// TIA Portal V17 export
// export: Created 2023-02-14T02:49:48.6840805Z, ExportSetting WithDefaults, DisplayName Totally Integrated Automation Portal, DisplayVersion V17, DisplayName TIA Portal Openness, DisplayVersion V17, DisplayName TIA Portal Teamcenter Gateway, DisplayVersion V17, DisplayName TIA Portal Version Control Interface, DisplayVersion V17, DisplayName SINAMICS Startdrive Advanced, DisplayVersion V17, DisplayName SINAMICS Startdrive G130, G150, S120, S150, SINAMICS MV, S210, DisplayVersion V17, DisplayName SINAMICS Startdrive G110M, G120, G120C, G120D, G120P, G115D, DisplayVersion V17, DisplayName STEP 7 Professional, DisplayVersion V17, DisplayName STEP 7 Safety, DisplayVersion V17, DisplayName WinCC Professional, DisplayVersion V17
FUNCTION_BLOCK "BFT_Type2"   // FB352, LAD
{ S7_Optimized_Access := 'TRUE' }
VERSION : 0.1
// Buffer Tank with Agitator
// stored: AutoNumber false, IsIECCheckEnabled false, IsRetainMemResEnabled false, MemoryReserve 100, SetENOAutomatically false, UDAEnableTagReadback false
   VAR_INPUT
      "IN_FBAV.01" : Bool := FALSE;   // Tank Flushing Water Valve
      "IN_FBAV.02" : Bool := FALSE;   // Tank CIP Top Inlet Valve
      "IN_FBAV.03" : Bool := FALSE;   // Tank Tank Outlet Valve
      "IN_FBAV.04" : Bool := FALSE;   // Tank CIP Return Valve
      "IN_FBAV.05" : Bool := FALSE;   // Tank Inlet Vinegar Valve
      "IN_FBAV.06" : Bool := FALSE;   // Tank CIP Valve
      "IN_FBAV.07" : Bool := FALSE;   // Tank CIP Valve
      "IN_FBAV.08" : Bool := FALSE;   // Line CIP Bypass Valve
      "IN_FBAV.09" : Bool := FALSE;   // Line CIP Valve
      "IN_FBAV.10" : Bool;   // Tank Inlet Valve
      "IN_FBAV.11" : Bool;   // Line CIP Valve
      "IN_FBAV.12" : Bool;   // Line CIP Valve
      IN_LT01 : Real;   // Tank Level Transmitter
      "IN_FBP.01" : Bool := FALSE;   // Transfer Pump
      "IN_P.01-Speed" : Real;   // Transfer Pump AV Speed
      "IN_FBP.02" : Bool := FALSE;   // CIP Pump
      "IN_P.02-Speed" : Real;   // CIP Pump AV Speed
      "IN_FBP.03" : Bool := FALSE;   // Supply Pump
      "IN_P.03-Speed" : Real;   // Supply Pump AV Speed
      IN_FBXA : Bool := FALSE;   // Agitator
      "IN_XA-Speed" : Real;   // Agitator AV Speed
      DosePumpSpeed : Real;
      "DoseON-OFF" : Bool := FALSE;
      "DosePumpON-OFF" : Bool := FALSE;
      CIPPulse : Bool := FALSE;
      CIP_Supply_ON : Bool;
      CIP_Busy : Bool;   // Line CIP in USE
      LineTrf_OK : Bool := FALSE;
      LineFlush_OK : Bool;
      Loading_Busy : Bool;   // Other tank at loading
      LCS_Start : Bool;   // Start Command from LCS
      LCS_Stop : Bool;   // Stop Command from LCS
      LCS_Dose : Bool;   // Start dose command from LCS
      InloadDose_AV : Bool;   // Inload Dose Valve Open
      InloadDose_P : Bool;   // Inload Dose Pump Running
      CountMode : Bool;   // 0 = Pulse Counting, 1 = Real Count
      FT_Pulse : Bool;   // Pulse Flow Meter
      FT_Total : Real;   // Inload Dose Actual Value
      IN_LDT : Date_And_Time;
   END_VAR
   VAR_OUTPUT
      "OUT_AV.01" : Bool := FALSE;   // Tank Flushing Water Valve
      "OUT_AV.02" : Bool := FALSE;   // Tank CIP Top Inlet Valve
      "OUT_AV.03" : Bool := FALSE;   // Tank Tank Outlet Valve
      "OUT_AV.04" : Bool := FALSE;   // Tank CIP Return Valve
      "OUT_AV.05" : Bool := FALSE;   // Tank Inlet Vinegar Valve
      "OUT_AV.06" : Bool := FALSE;   // Tank CIP Valve
      "OUT_AV.07" : Bool := FALSE;   // Tank CIP Valve
      "OUT_AV.08" : Bool := FALSE;   // Line CIP Bypass Valve
      "OUT_AV.09" : Bool := FALSE;   // Line CIP Valve
      "OUT_AV.10" : Bool;   // Tank Inlet Valve
      "OUT_AV.11" : Bool;   // Line CIP Valve
      "OUT_AV.12" : Bool;   // Line CIP Valve
      "OUT_P.01" : Bool := FALSE;   // Transfer Pump
      "OUT_P.01-Speed" : Real;   // Transfer Pump AV Speed
      "OUT_P.02" : Bool := FALSE;   // CIP Pump
      "OUT_P.02-Speed" : Real;   // CIP Pump AV Speed
      "OUT_P.03" : Bool := FALSE;   // Supply Pump
      "OUT_P.03-Speed" : Real;   // Supply Pump AV Speed
      OUT_XA : Bool := FALSE;   // Agitator
      "OUT_XA-Speed" : Real;   // Agitator AV Speed
      OUT_InloadDose_Idle : Bool;   // Inload Dose Idle State
      OUT_InloadDose_AV : Bool;   // Inload Dose Valve Cmd Open
      OUT_InloadDose_P : Bool;   // Inload Dose Pump Cmd Running
      OUT_InloadDose_P_Speed : Real;   // Inload Dose Pump SP Speed
      OUT_CIPTank_AVOpen : Bool;
      OUT_CIPLine_AVOpen : Bool;
   END_VAR
   VAR
      Cmd { ExternalAccessible := 'False'; ExternalVisible := 'False'; ExternalWritable := 'False'} : Struct
         Inload { ExternalAccessible := 'False'; ExternalVisible := 'False'; ExternalWritable := 'False'} : Bool;   // Start Loading
         Dose_start { ExternalAccessible := 'False'; ExternalVisible := 'False'; ExternalWritable := 'False'} : Bool;   // Start dose
         Dose_pause { ExternalAccessible := 'False'; ExternalVisible := 'False'; ExternalWritable := 'False'} : Bool;   // Pause dose
         RaadyForMix { ExternalAccessible := 'False'; ExternalVisible := 'False'; ExternalWritable := 'False'} : Bool;   // Tank Ready for Blending
         Tank_CIP_Req { ExternalAccessible := 'False'; ExternalVisible := 'False'; ExternalWritable := 'False'} : Bool;
         Line_CIP_Req { ExternalAccessible := 'False'; ExternalVisible := 'False'; ExternalWritable := 'False'} : Bool;
         Flushing { ExternalAccessible := 'False'; ExternalVisible := 'False'; ExternalWritable := 'False'} : Bool;   // Water Flushing
         Flush_Select { ExternalAccessible := 'False'; ExternalVisible := 'False'; ExternalWritable := 'False'} : Byte;
         Agitator_Mode { ExternalAccessible := 'False'; ExternalVisible := 'False'; ExternalWritable := 'False'} : Bool;   // 0 = Auto
         Agitator_Man_ONOFF { ExternalAccessible := 'False'; ExternalVisible := 'False'; ExternalWritable := 'False'} : Bool;
         Agitator_SpeedMode { ExternalAccessible := 'False'; ExternalVisible := 'False'; ExternalWritable := 'False'} : Bool;   // 0 = Fix SP ; 1 = Level
      END_STRUCT;
      Param { ExternalAccessible := 'False'; ExternalVisible := 'False'; ExternalWritable := 'False'} : Struct
         SP_Level_LL { ExternalAccessible := 'False'; ExternalVisible := 'False'; ExternalWritable := 'False'} : Real := 10.0;
         SP_Level_ML { ExternalAccessible := 'False'; ExternalVisible := 'False'; ExternalWritable := 'False'} : Real := 80.0;
         SP_Level_HL { ExternalAccessible := 'False'; ExternalVisible := 'False'; ExternalWritable := 'False'} : Real := 100.0;
         SP_Level_Agi_ON1 { ExternalAccessible := 'False'; ExternalVisible := 'False'; ExternalWritable := 'False'} : Real := 20.0;   // product level over from lower blade
         SP_Level_Agi_OFF1 { ExternalAccessible := 'False'; ExternalVisible := 'False'; ExternalWritable := 'False'} : Real := 60.0;   // product level almost from mid blade
         SP_Level_Agi_ON2 { ExternalAccessible := 'False'; ExternalVisible := 'False'; ExternalWritable := 'False'} : Real := 62.0;   // product level over from mid blade
         SP_Level_Agi_OFF2 { ExternalAccessible := 'False'; ExternalVisible := 'False'; ExternalWritable := 'False'} : Real := 80.0;   // product level almost from upper blade
         SP_Level_Agi_ON3 { ExternalAccessible := 'False'; ExternalVisible := 'False'; ExternalWritable := 'False'} : Real := 82.0;   // product level over from upper blade
         SupplyPump_SP_Speed { ExternalAccessible := 'False'; ExternalVisible := 'False'; ExternalWritable := 'False'} : Real := 80.0;   // Inload Pump SP Speed
         Agitator_SP_Speed { ExternalAccessible := 'False'; ExternalVisible := 'False'; ExternalWritable := 'False'} : Real := 80.0;   // Agitator SP Speed
         RawDose_SP_Qty { ExternalAccessible := 'False'; ExternalVisible := 'False'; ExternalWritable := 'False'} : Real := 300.0;   // Raw Matrial Dose_SP Quantity
         RawDose_Fine_Qty { ExternalAccessible := 'False'; ExternalVisible := 'False'; ExternalWritable := 'False'} : Real := 20.0;   // Raw Matrial Dose_Fine Quantity Percen
         RawDose_Stop_Qty { ExternalAccessible := 'False'; ExternalVisible := 'False'; ExternalWritable := 'False'} : Real := 0.01;   // Raw Matrial Dose_Stop Quantity Percen
         RawDose_SP_Speed { ExternalAccessible := 'False'; ExternalVisible := 'False'; ExternalWritable := 'False'} : Real := 80.0;   // Raw Matrial Dose_SP Speed
         RawDose_Fine_Speed { ExternalAccessible := 'False'; ExternalVisible := 'False'; ExternalWritable := 'False'} : Real := 20.0;   // Raw Matrial Dose_Fine Speed
         L_Hi_Lim { ExternalAccessible := 'False'; ExternalVisible := 'False'; ExternalWritable := 'False'} : Real := 100.0;
         L_Lo_Lim { ExternalAccessible := 'False'; ExternalVisible := 'False'; ExternalWritable := 'False'} : Real := 0.0;
         L_Hys { ExternalAccessible := 'False'; ExternalVisible := 'False'; ExternalWritable := 'False'} : Real := 5.0;
         FlushingTime { ExternalAccessible := 'False'; ExternalVisible := 'False'; ExternalWritable := 'False'} : Time := T#10s;
         CIP_Trf_SP_Speed { ExternalAccessible := 'False'; ExternalVisible := 'False'; ExternalWritable := 'False'} : Real := 80.0;
         CIP_Ret_ON_SP { ExternalAccessible := 'False'; ExternalVisible := 'False'; ExternalWritable := 'False'} : Real := 5.0;
         CIP_Ret_OFF_SP { ExternalAccessible := 'False'; ExternalVisible := 'False'; ExternalWritable := 'False'} : Real;
      END_STRUCT;
      State { ExternalAccessible := 'False'; ExternalVisible := 'False'; ExternalWritable := 'False'} : Struct   // Tank in loading state
         Tank_inloading { ExternalAccessible := 'False'; ExternalVisible := 'False'; ExternalWritable := 'False'} : Bool;
         Tank_inRawDose { ExternalAccessible := 'False'; ExternalVisible := 'False'; ExternalWritable := 'False'} : Bool;
         Tank_inCIP { ExternalAccessible := 'False'; ExternalVisible := 'False'; ExternalWritable := 'False'} : Bool;
         Line_inCIP { ExternalAccessible := 'False'; ExternalVisible := 'False'; ExternalWritable := 'False'} : Bool;
         Flushing { ExternalAccessible := 'False'; ExternalVisible := 'False'; ExternalWritable := 'False'} : Bool;
         Tank_LL { ExternalAccessible := 'False'; ExternalVisible := 'False'; ExternalWritable := 'False'} : Bool;
         Tank_ML { ExternalAccessible := 'False'; ExternalVisible := 'False'; ExternalWritable := 'False'} : Bool;
         Tank_HL { ExternalAccessible := 'False'; ExternalVisible := 'False'; ExternalWritable := 'False'} : Bool;
         L_Agi_ON1 { ExternalAccessible := 'False'; ExternalVisible := 'False'; ExternalWritable := 'False'} : Bool;   // Lower Blade
         L_Agi_ON2 { ExternalAccessible := 'False'; ExternalVisible := 'False'; ExternalWritable := 'False'} : Bool;   // Midle Blade
         L_Agi_ON3 { ExternalAccessible := 'False'; ExternalVisible := 'False'; ExternalWritable := 'False'} : Bool;   // Upper Blade
         Inload_Enable { ExternalAccessible := 'False'; ExternalVisible := 'False'; ExternalWritable := 'False'} : Bool;
         Tank_CIP_Enable { ExternalAccessible := 'False'; ExternalVisible := 'False'; ExternalWritable := 'False'} : Bool;
         Line_CIP_Enable { ExternalAccessible := 'False'; ExternalVisible := 'False'; ExternalWritable := 'False'} : Bool;
         Flushing_Enable { ExternalAccessible := 'False'; ExternalVisible := 'False'; ExternalWritable := 'False'} : Bool;
         Flush_selected { ExternalAccessible := 'False'; ExternalVisible := 'False'; ExternalWritable := 'False'} : Byte;
         CIP_Request_OK { ExternalAccessible := 'False'; ExternalVisible := 'False'; ExternalWritable := 'False'} : Bool;
         CIP_ReturnON { ExternalAccessible := 'False'; ExternalVisible := 'False'; ExternalWritable := 'False'} : Bool;
         Ready_For_Transfer_EN { ExternalAccessible := 'False'; ExternalVisible := 'False'; ExternalWritable := 'False'} : Bool;   // Tank Ready for Transfer to Blending
         Ready_For_Transfer { ExternalAccessible := 'False'; ExternalVisible := 'False'; ExternalWritable := 'False'} : Bool;   // Tank Ready for Transfer to Blending
         Transfer_to_Blend { ExternalAccessible := 'False'; ExternalVisible := 'False'; ExternalWritable := 'False'} : Bool;
         HWT_Status { ExternalAccessible := 'False'; ExternalVisible := 'False'; ExternalWritable := 'False'} : Int;
      END_STRUCT;
      alwaysON : Bool;
      L_Hys_Abs : Real;
      Hys_Level_HL : Real;
      Hys_Level_ML : Real;
      Hys_Level_LL : Real;
      RawDose_Stop_Qty : Real;
      "FT Counter" : Real;
      "Pulse/Liter" : Real := 1.0;
      AwalTolaizer { S7_SetPoint := 'True'} : Real;
      AkhirTolaizer : Real;
      TargetTotalizer : Real;
      r : Struct
         PosE1 : Bool;
         PosE2 : Bool;
         PosE3 : Bool;
         PosE4 : Bool;
         PosE5 : Bool;
         PosE6 : Bool;
         PosE7 : Bool;
         PosE8 : Bool;
         PosE9 : Bool;
         PosE10 : Bool;
         PosE11 : Bool;
         PosE12 : Bool;
         PosE13 : Bool;
         PosE14 : Bool;
         PosE15 : Bool;
         PosE16 : Bool;
         PosE17 : Bool;
         PosE18 : Bool;
         PosE19 : Bool;
         PosE20 : Bool;
         PosE21 : Bool;
         PosE22 : Bool;
         PosE23 : Bool;
         PosE24 : Bool;
         PosE25 : Bool;
         PosE26 : Bool;
         PosE27 : Bool;
         PosE28 : Bool;
         PosE29 : Bool;
         PosE30 : Bool;
         PosE31 : Bool;
         PosE32 : Bool;
      END_STRUCT;
      Actuator : Struct
         AV_Outlet : Bool;
         TransferPump : Bool;
         FlushPump : Bool;
         CV_Steam : Bool;
         Pump : Bool;
         Agitator_level : Bool;
         LCS_OnOff : Bool;
      END_STRUCT;
      FlushingTim : TON_TIME;
      SPumpTim { S7_SetPoint := 'True'} : TON_TIME;
      AVinloadTim { S7_SetPoint := 'True'} : TON_TIME;
      L_AgiTim { S7_SetPoint := 'True'} : TON_TIME;
      Dose { S7_SetPoint := 'True'} : "DOSE";
   END_VAR
   VAR_TEMP   // added for the SCL form of the ladder/FBD networks
      _w1 : Bool;
      _w2 : Bool;
      _w3 : Bool;
      _w4 : Bool;
      _w5 : Bool;
      _w6 : Bool;
   END_VAR
BEGIN

REGION Network 1: Always_ON
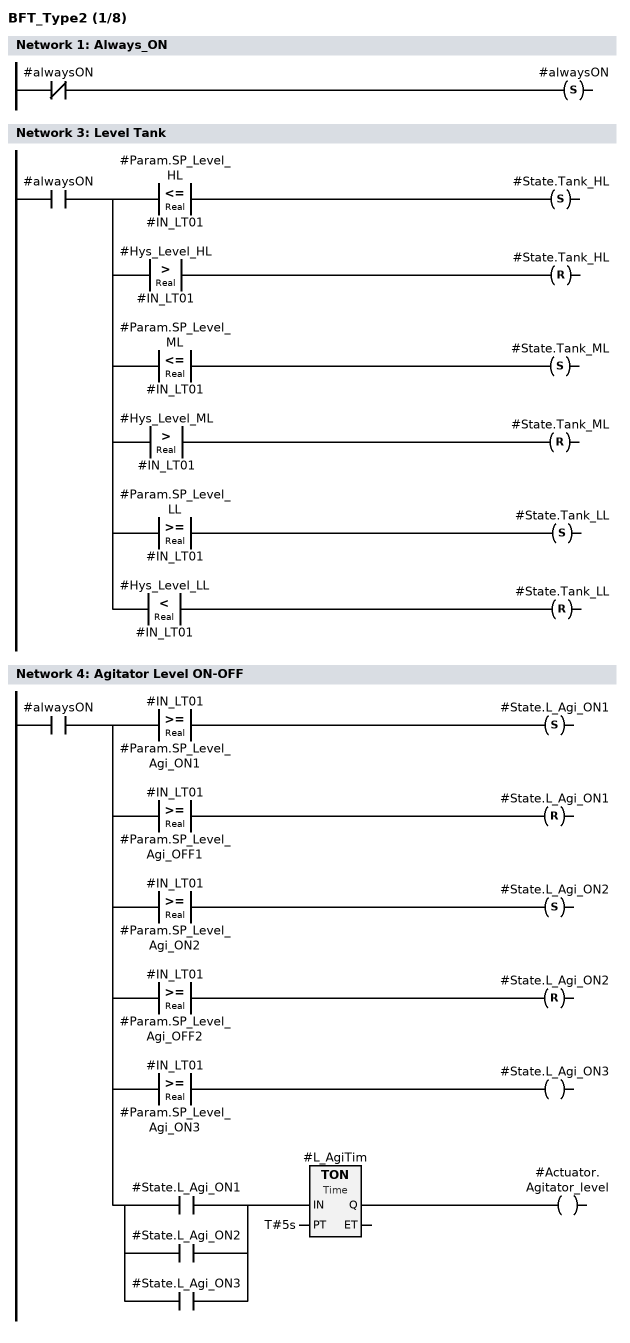
   RUNG wire#powerrail
      I_Contact( #alwaysON )
      S_Coil( #alwaysON )
   END_RUNG
   // the same network as SCL:
   IF NOT #alwaysON THEN #alwaysON := TRUE; END_IF;
END_REGION

NETWORK
TITLE = Hys Calculation
//Level Hys Absolute
      L     #Param.L_Hi_Lim;
      L     #Param.L_Lo_Lim;
      -R;
      L     100.0;
      /R;
      L     #Param.L_Hys;
      *R;
      T     #L_Hys_Abs;
//Tank High Level
      L     #Param.SP_Level_HL;
      L     #L_Hys_Abs;
      -R;
      T     #Hys_Level_HL;
//Tank Mid Level
      L     #Param.SP_Level_ML;
      L     #L_Hys_Abs;
      -R;
      T     #Hys_Level_ML;
//Tank Low Level
      L     #Param.SP_Level_LL;
      L     #L_Hys_Abs;
      +R;
      T     #Hys_Level_LL;


REGION Network 3: Level Tank
   RUNG wire#powerrail
      Contact( #alwaysON )
      wire#w1
      { S7_Templates := "SrcType := Real" } LE_Contact(in1 := #Param.SP_Level_HL, in2 := #IN_LT01)
      S_Coil( #State.Tank_HL )
   END_RUNG
   RUNG wire#w1
      { S7_Templates := "SrcType := Real" } GT_Contact(in1 := #Hys_Level_HL, in2 := #IN_LT01)
      R_Coil( #State.Tank_HL )
   END_RUNG
   RUNG wire#w1
      { S7_Templates := "SrcType := Real" } LE_Contact(in1 := #Param.SP_Level_ML, in2 := #IN_LT01)
      S_Coil( #State.Tank_ML )
   END_RUNG
   RUNG wire#w1
      { S7_Templates := "SrcType := Real" } GT_Contact(in1 := #Hys_Level_ML, in2 := #IN_LT01)
      R_Coil( #State.Tank_ML )
   END_RUNG
   RUNG wire#w1
      { S7_Templates := "SrcType := Real" } GE_Contact(in1 := #Param.SP_Level_LL, in2 := #IN_LT01)
      S_Coil( #State.Tank_LL )
   END_RUNG
   RUNG wire#w1
      { S7_Templates := "SrcType := Real" } LT_Contact(in1 := #Hys_Level_LL, in2 := #IN_LT01)
      R_Coil( #State.Tank_LL )
   END_RUNG
   // the same network as SCL:
   IF #alwaysON AND (#Param.SP_Level_HL <= #IN_LT01) THEN #State.Tank_HL := TRUE; END_IF;
   IF #alwaysON AND (#Hys_Level_HL > #IN_LT01) THEN #State.Tank_HL := FALSE; END_IF;
   IF #alwaysON AND (#Param.SP_Level_ML <= #IN_LT01) THEN #State.Tank_ML := TRUE; END_IF;
   IF #alwaysON AND (#Hys_Level_ML > #IN_LT01) THEN #State.Tank_ML := FALSE; END_IF;
   IF #alwaysON AND (#Param.SP_Level_LL >= #IN_LT01) THEN #State.Tank_LL := TRUE; END_IF;
   IF #alwaysON AND (#Hys_Level_LL < #IN_LT01) THEN #State.Tank_LL := FALSE; END_IF;
END_REGION

REGION Network 4: Agitator Level ON-OFF
   RUNG wire#powerrail
      Contact( #alwaysON )
      wire#w1
      { S7_Templates := "SrcType := Real" } GE_Contact(in1 := #IN_LT01, in2 := #Param.SP_Level_Agi_ON1)
      S_Coil( #State.L_Agi_ON1 )
   END_RUNG
   RUNG wire#w1
      { S7_Templates := "SrcType := Real" } GE_Contact(in1 := #IN_LT01, in2 := #Param.SP_Level_Agi_OFF1)
      R_Coil( #State.L_Agi_ON1 )
   END_RUNG
   RUNG wire#w1
      { S7_Templates := "SrcType := Real" } GE_Contact(in1 := #IN_LT01, in2 := #Param.SP_Level_Agi_ON2)
      S_Coil( #State.L_Agi_ON2 )
   END_RUNG
   RUNG wire#w1
      { S7_Templates := "SrcType := Real" } GE_Contact(in1 := #IN_LT01, in2 := #Param.SP_Level_Agi_OFF2)
      R_Coil( #State.L_Agi_ON2 )
   END_RUNG
   RUNG wire#w1
      { S7_Templates := "SrcType := Real" } GE_Contact(in1 := #IN_LT01, in2 := #Param.SP_Level_Agi_ON3)
      Coil( #State.L_Agi_ON3 )
   END_RUNG
   RUNG wire#w1
      Contact( #State.L_Agi_ON1 )
      wire#w2
      { S7_Templates := "time_type := Time" } #L_AgiTim.TON(pt := T#5s, et =>)
      Coil( #Actuator.Agitator_level )
   END_RUNG
   RUNG wire#w1
      Contact( #State.L_Agi_ON2 )
   END_RUNG wire#w2
   RUNG wire#w1
      Contact( #State.L_Agi_ON3 )
   END_RUNG wire#w2
   // the same network as SCL:
   IF #alwaysON AND (#IN_LT01 >= #Param.SP_Level_Agi_ON1) THEN #State.L_Agi_ON1 := TRUE; END_IF;
   IF #alwaysON AND (#IN_LT01 >= #Param.SP_Level_Agi_OFF1) THEN #State.L_Agi_ON1 := FALSE; END_IF;
   IF #alwaysON AND (#IN_LT01 >= #Param.SP_Level_Agi_ON2) THEN #State.L_Agi_ON2 := TRUE; END_IF;
   IF #alwaysON AND (#IN_LT01 >= #Param.SP_Level_Agi_OFF2) THEN #State.L_Agi_ON2 := FALSE; END_IF;
   #State.L_Agi_ON3 := #alwaysON AND (#IN_LT01 >= #Param.SP_Level_Agi_ON3);
   #L_AgiTim(IN := #alwaysON AND (#State.L_Agi_ON1 OR #State.L_Agi_ON2 OR #State.L_Agi_ON3), PT := T#5s);   // TON
   #Actuator.Agitator_level := #L_AgiTim.Q;
END_REGION

REGION Network 5: Reset Command Inload
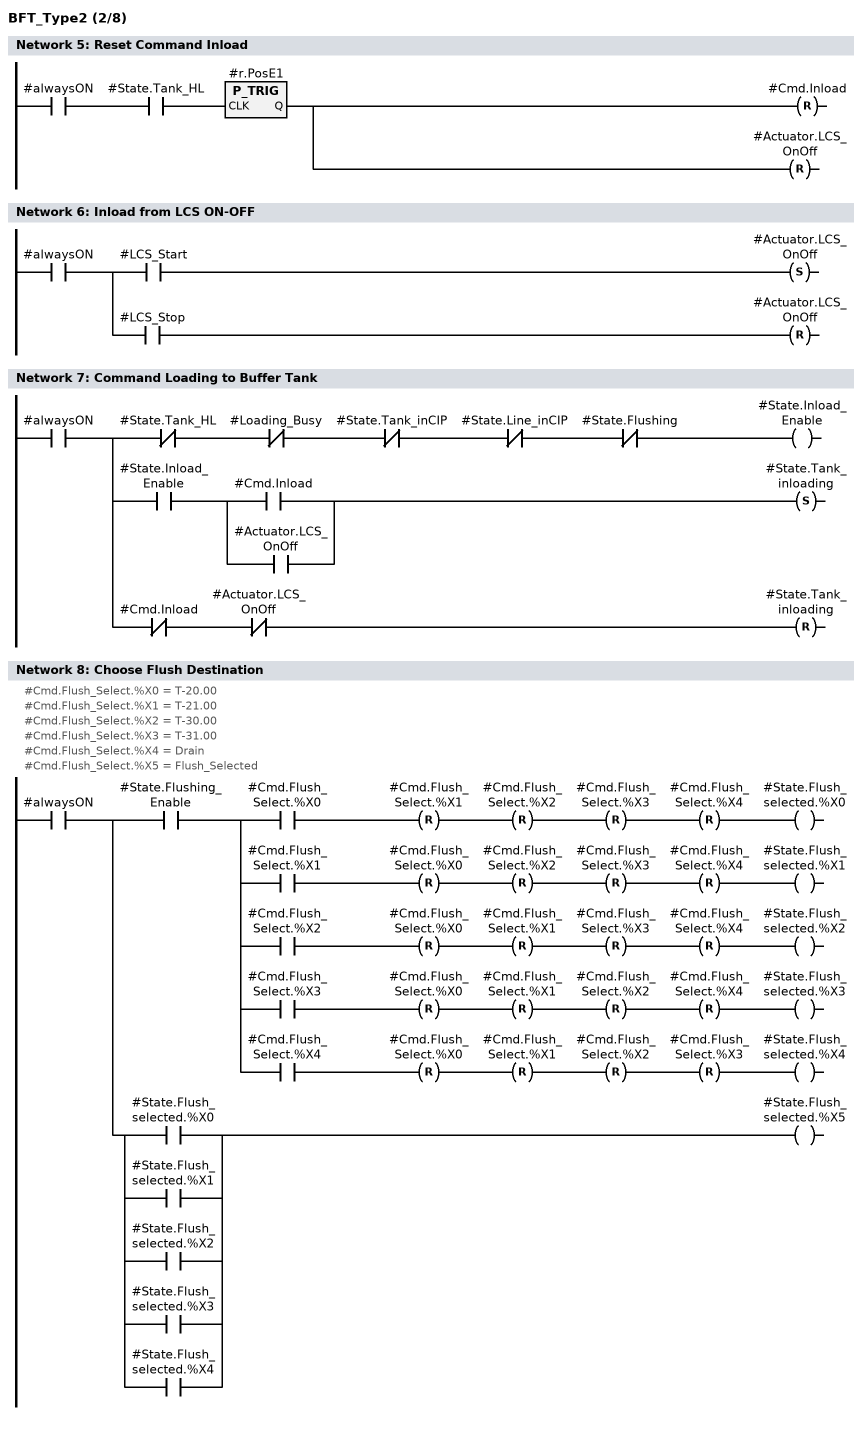
   RUNG wire#powerrail
      Contact( #alwaysON )
      Contact( #State.Tank_HL )
      P_Trig( #r.PosE1 )
      wire#w1
      R_Coil( #Cmd.Inload )
   END_RUNG
   RUNG wire#w1
      R_Coil( #Actuator.LCS_OnOff )
   END_RUNG
   // the same network as SCL:
   #_w1 := #alwaysON AND #State.Tank_HL;
   #_w2 := #_w1 AND NOT #r.PosE1;   // rising edge
   #r.PosE1 := #_w1;
   IF #_w2 THEN
       #Cmd.Inload := FALSE;
       #Actuator.LCS_OnOff := FALSE;
   END_IF;
END_REGION

REGION Network 6: Inload from LCS ON-OFF
   RUNG wire#powerrail
      Contact( #alwaysON )
      wire#w1
      Contact( #LCS_Start )
      S_Coil( #Actuator.LCS_OnOff )
   END_RUNG
   RUNG wire#w1
      Contact( #LCS_Stop )
      R_Coil( #Actuator.LCS_OnOff )
   END_RUNG
   // the same network as SCL:
   IF #alwaysON AND #LCS_Start THEN #Actuator.LCS_OnOff := TRUE; END_IF;
   IF #alwaysON AND #LCS_Stop THEN #Actuator.LCS_OnOff := FALSE; END_IF;
END_REGION

REGION Network 7: Command Loading to Buffer Tank
   RUNG wire#powerrail
      Contact( #alwaysON )
      wire#w1
      I_Contact( #State.Tank_HL )
      I_Contact( #Loading_Busy )
      I_Contact( #State.Tank_inCIP )
      I_Contact( #State.Line_inCIP )
      I_Contact( #State.Flushing )
      Coil( #State.Inload_Enable )
   END_RUNG
   RUNG wire#w1
      Contact( #State.Inload_Enable )
      wire#w2
      Contact( #Cmd.Inload )
      wire#w3
      S_Coil( #State.Tank_inloading )
   END_RUNG
   RUNG wire#w2
      Contact( #Actuator.LCS_OnOff )
   END_RUNG wire#w3
   RUNG wire#w1
      I_Contact( #Cmd.Inload )
      I_Contact( #Actuator.LCS_OnOff )
      R_Coil( #State.Tank_inloading )
   END_RUNG
   // the same network as SCL:
   #State.Inload_Enable := #alwaysON AND NOT #State.Tank_HL AND NOT #Loading_Busy AND NOT #State.Tank_inCIP AND NOT #State.Line_inCIP AND NOT #State.Flushing;
   IF #alwaysON AND #State.Inload_Enable AND (#Cmd.Inload OR #Actuator.LCS_OnOff) THEN
       #State.Tank_inloading := TRUE;
   END_IF;
   IF #alwaysON AND NOT #Cmd.Inload AND NOT #Actuator.LCS_OnOff THEN #State.Tank_inloading := FALSE; END_IF;
END_REGION

REGION Network 8: Choose Flush Destination
   // #Cmd.Flush_Select.%X0 = T-20.00
   // #Cmd.Flush_Select.%X1 = T-21.00
   // #Cmd.Flush_Select.%X2 = T-30.00
   // #Cmd.Flush_Select.%X3 = T-31.00
   // #Cmd.Flush_Select.%X4 = Drain
   // #Cmd.Flush_Select.%X5 = Flush_Selected
   RUNG wire#powerrail
      Contact( #alwaysON )
      wire#w1
      Contact( #State.Flushing_Enable )
      wire#w2
      Contact( #Cmd.Flush_Select.%X0 )
      R_Coil( #Cmd.Flush_Select.%X1 )
      R_Coil( #Cmd.Flush_Select.%X2 )
      R_Coil( #Cmd.Flush_Select.%X3 )
      R_Coil( #Cmd.Flush_Select.%X4 )
      Coil( #State.Flush_selected.%X0 )
   END_RUNG
   RUNG wire#w2
      Contact( #Cmd.Flush_Select.%X1 )
      R_Coil( #Cmd.Flush_Select.%X0 )
      R_Coil( #Cmd.Flush_Select.%X2 )
      R_Coil( #Cmd.Flush_Select.%X3 )
      R_Coil( #Cmd.Flush_Select.%X4 )
      Coil( #State.Flush_selected.%X1 )
   END_RUNG
   RUNG wire#w2
      Contact( #Cmd.Flush_Select.%X2 )
      R_Coil( #Cmd.Flush_Select.%X0 )
      R_Coil( #Cmd.Flush_Select.%X1 )
      R_Coil( #Cmd.Flush_Select.%X3 )
      R_Coil( #Cmd.Flush_Select.%X4 )
      Coil( #State.Flush_selected.%X2 )
   END_RUNG
   RUNG wire#w2
      Contact( #Cmd.Flush_Select.%X3 )
      R_Coil( #Cmd.Flush_Select.%X0 )
      R_Coil( #Cmd.Flush_Select.%X1 )
      R_Coil( #Cmd.Flush_Select.%X2 )
      R_Coil( #Cmd.Flush_Select.%X4 )
      Coil( #State.Flush_selected.%X3 )
   END_RUNG
   RUNG wire#w2
      Contact( #Cmd.Flush_Select.%X4 )
      R_Coil( #Cmd.Flush_Select.%X0 )
      R_Coil( #Cmd.Flush_Select.%X1 )
      R_Coil( #Cmd.Flush_Select.%X2 )
      R_Coil( #Cmd.Flush_Select.%X3 )
      Coil( #State.Flush_selected.%X4 )
   END_RUNG
   RUNG wire#w1
      Contact( #State.Flush_selected.%X0 )
      wire#w3
      Coil( #State.Flush_selected.%X5 )
   END_RUNG
   RUNG wire#w1
      Contact( #State.Flush_selected.%X1 )
   END_RUNG wire#w3
   RUNG wire#w1
      Contact( #State.Flush_selected.%X2 )
   END_RUNG wire#w3
   RUNG wire#w1
      Contact( #State.Flush_selected.%X3 )
   END_RUNG wire#w3
   RUNG wire#w1
      Contact( #State.Flush_selected.%X4 )
   END_RUNG wire#w3
   // the same network as SCL:
   #_w1 := #alwaysON AND #State.Flushing_Enable;
   #_w2 := #_w1 AND #Cmd.Flush_Select.%X0;
   IF #_w2 THEN
       #Cmd.Flush_Select.%X1 := FALSE;
       #Cmd.Flush_Select.%X2 := FALSE;
       #Cmd.Flush_Select.%X3 := FALSE;
       #Cmd.Flush_Select.%X4 := FALSE;
   END_IF;
   #State.Flush_selected.%X0 := #_w2;
   #_w3 := #_w1 AND #Cmd.Flush_Select.%X1;
   IF #_w3 THEN
       #Cmd.Flush_Select.%X0 := FALSE;
       #Cmd.Flush_Select.%X2 := FALSE;
       #Cmd.Flush_Select.%X3 := FALSE;
       #Cmd.Flush_Select.%X4 := FALSE;
   END_IF;
   #State.Flush_selected.%X1 := #_w3;
   #_w4 := #_w1 AND #Cmd.Flush_Select.%X2;
   IF #_w4 THEN
       #Cmd.Flush_Select.%X0 := FALSE;
       #Cmd.Flush_Select.%X1 := FALSE;
       #Cmd.Flush_Select.%X3 := FALSE;
       #Cmd.Flush_Select.%X4 := FALSE;
   END_IF;
   #State.Flush_selected.%X2 := #_w4;
   #_w5 := #_w1 AND #Cmd.Flush_Select.%X3;
   IF #_w5 THEN
       #Cmd.Flush_Select.%X0 := FALSE;
       #Cmd.Flush_Select.%X1 := FALSE;
       #Cmd.Flush_Select.%X2 := FALSE;
       #Cmd.Flush_Select.%X4 := FALSE;
   END_IF;
   #State.Flush_selected.%X3 := #_w5;
   #_w6 := #_w1 AND #Cmd.Flush_Select.%X4;
   IF #_w6 THEN
       #Cmd.Flush_Select.%X0 := FALSE;
       #Cmd.Flush_Select.%X1 := FALSE;
       #Cmd.Flush_Select.%X2 := FALSE;
       #Cmd.Flush_Select.%X3 := FALSE;
   END_IF;
   #State.Flush_selected.%X4 := #_w6;
   #State.Flush_selected.%X5 := #alwaysON AND (#State.Flush_selected.%X0 OR #State.Flush_selected.%X1 OR #State.Flush_selected.%X2 OR #State.Flush_selected.%X3 OR #State.Flush_selected.%X4);
END_REGION

REGION Network 9: Command Water Flushing
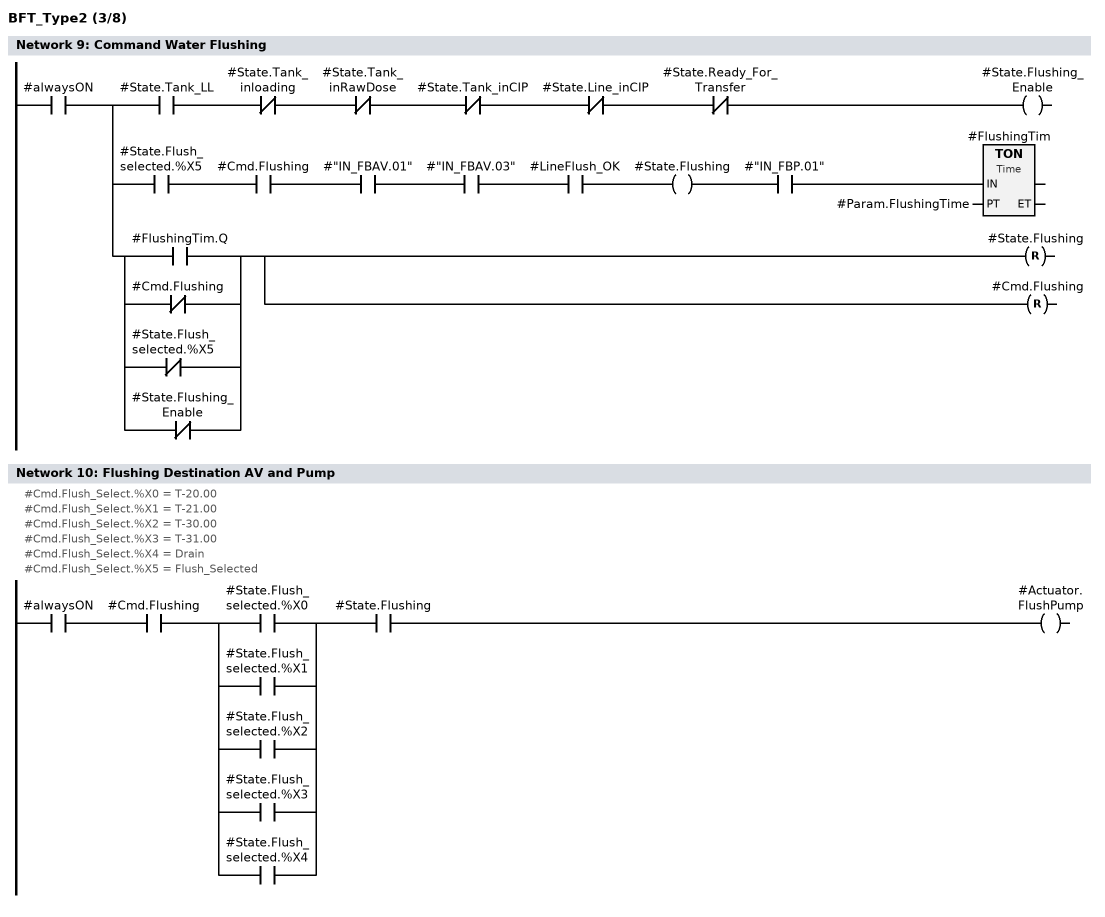
   RUNG wire#powerrail
      Contact( #alwaysON )
      wire#w1
      Contact( #State.Tank_LL )
      I_Contact( #State.Tank_inloading )
      I_Contact( #State.Tank_inRawDose )
      I_Contact( #State.Tank_inCIP )
      I_Contact( #State.Line_inCIP )
      I_Contact( #State.Ready_For_Transfer )
      Coil( #State.Flushing_Enable )
   END_RUNG
   RUNG wire#w1
      Contact( #State.Flush_selected.%X5 )
      Contact( #Cmd.Flushing )
      Contact( #"IN_FBAV.01" )
      Contact( #"IN_FBAV.03" )
      Contact( #LineFlush_OK )
      Coil( #State.Flushing )
      Contact( #"IN_FBP.01" )
      { S7_Templates := "time_type := Time" } #FlushingTim.TON(pt := #Param.FlushingTime, et =>)
   END_RUNG
   RUNG wire#w1
      Contact( #FlushingTim.Q )
      wire#w2
      R_Coil( #State.Flushing )
   END_RUNG
   RUNG wire#w1
      I_Contact( #Cmd.Flushing )
   END_RUNG wire#w2
   RUNG wire#w1
      I_Contact( #State.Flush_selected.%X5 )
   END_RUNG wire#w2
   RUNG wire#w1
      I_Contact( #State.Flushing_Enable )
   END_RUNG wire#w2
   RUNG wire#w2
      R_Coil( #Cmd.Flushing )
   END_RUNG
   // the same network as SCL:
   #State.Flushing_Enable := #alwaysON AND #State.Tank_LL AND NOT #State.Tank_inloading AND NOT #State.Tank_inRawDose AND NOT #State.Tank_inCIP AND NOT #State.Line_inCIP AND NOT #State.Ready_For_Transfer;
   #State.Flushing := #alwaysON AND #State.Flush_selected.%X5 AND #Cmd.Flushing AND #"IN_FBAV.01" AND #"IN_FBAV.03" AND #LineFlush_OK;
   #FlushingTim(IN := #State.Flushing AND #"IN_FBP.01", PT := #Param.FlushingTime);   // TON
   IF #alwaysON AND (#FlushingTim.Q OR NOT #Cmd.Flushing OR NOT #State.Flush_selected.%X5 OR NOT #State.Flushing_Enable) THEN
       #State.Flushing := FALSE;
       #Cmd.Flushing := FALSE;
   END_IF;
END_REGION

REGION Network 10: Flushing Destination AV and Pump
   // #Cmd.Flush_Select.%X0 = T-20.00
   // #Cmd.Flush_Select.%X1 = T-21.00
   // #Cmd.Flush_Select.%X2 = T-30.00
   // #Cmd.Flush_Select.%X3 = T-31.00
   // #Cmd.Flush_Select.%X4 = Drain
   // #Cmd.Flush_Select.%X5 = Flush_Selected
   RUNG wire#powerrail
      Contact( #alwaysON )
      Contact( #Cmd.Flushing )
      wire#w1
      Contact( #State.Flush_selected.%X0 )
      wire#w2
      Contact( #State.Flushing )
      Coil( #Actuator.FlushPump )
   END_RUNG
   RUNG wire#w1
      Contact( #State.Flush_selected.%X1 )
   END_RUNG wire#w2
   RUNG wire#w1
      Contact( #State.Flush_selected.%X2 )
   END_RUNG wire#w2
   RUNG wire#w1
      Contact( #State.Flush_selected.%X3 )
   END_RUNG wire#w2
   RUNG wire#w1
      Contact( #State.Flush_selected.%X4 )
   END_RUNG wire#w2
   // the same network as SCL:
   #Actuator.FlushPump := #alwaysON AND #Cmd.Flushing AND (#State.Flush_selected.%X0 OR #State.Flush_selected.%X1 OR #State.Flush_selected.%X2 OR #State.Flush_selected.%X3 OR #State.Flush_selected.%X4) AND #State.Flushing;
END_REGION

REGION Network 11: Command CIP
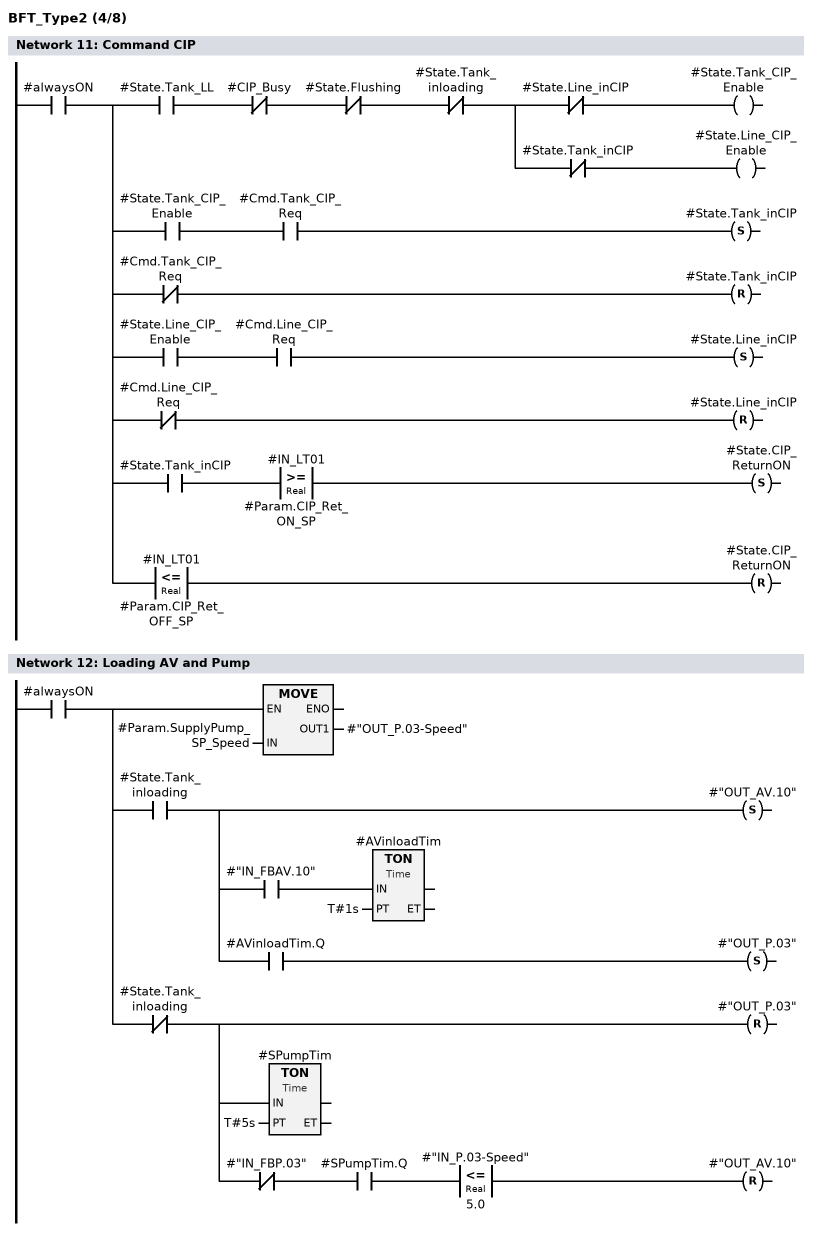
   RUNG wire#powerrail
      Contact( #alwaysON )
      wire#w1
      Contact( #State.Tank_LL )
      I_Contact( #CIP_Busy )
      I_Contact( #State.Flushing )
      I_Contact( #State.Tank_inloading )
      wire#w2
      I_Contact( #State.Line_inCIP )
      Coil( #State.Tank_CIP_Enable )
   END_RUNG
   RUNG wire#w2
      I_Contact( #State.Tank_inCIP )
      Coil( #State.Line_CIP_Enable )
   END_RUNG
   RUNG wire#w1
      Contact( #State.Tank_CIP_Enable )
      Contact( #Cmd.Tank_CIP_Req )
      S_Coil( #State.Tank_inCIP )
   END_RUNG
   RUNG wire#w1
      I_Contact( #Cmd.Tank_CIP_Req )
      R_Coil( #State.Tank_inCIP )
   END_RUNG
   RUNG wire#w1
      Contact( #State.Line_CIP_Enable )
      Contact( #Cmd.Line_CIP_Req )
      S_Coil( #State.Line_inCIP )
   END_RUNG
   RUNG wire#w1
      I_Contact( #Cmd.Line_CIP_Req )
      R_Coil( #State.Line_inCIP )
   END_RUNG
   RUNG wire#w1
      Contact( #State.Tank_inCIP )
      { S7_Templates := "SrcType := Real" } GE_Contact(in1 := #IN_LT01, in2 := #Param.CIP_Ret_ON_SP)
      S_Coil( #State.CIP_ReturnON )
   END_RUNG
   RUNG wire#w1
      { S7_Templates := "SrcType := Real" } LE_Contact(in1 := #IN_LT01, in2 := #Param.CIP_Ret_OFF_SP)
      R_Coil( #State.CIP_ReturnON )
   END_RUNG
   // the same network as SCL:
   #_w1 := #alwaysON AND #State.Tank_LL AND NOT #CIP_Busy AND NOT #State.Flushing AND NOT #State.Tank_inloading;
   #State.Tank_CIP_Enable := #_w1 AND NOT #State.Line_inCIP;
   #State.Line_CIP_Enable := #_w1 AND NOT #State.Tank_inCIP;
   IF #alwaysON AND #State.Tank_CIP_Enable AND #Cmd.Tank_CIP_Req THEN #State.Tank_inCIP := TRUE; END_IF;
   IF #alwaysON AND NOT #Cmd.Tank_CIP_Req THEN #State.Tank_inCIP := FALSE; END_IF;
   IF #alwaysON AND #State.Line_CIP_Enable AND #Cmd.Line_CIP_Req THEN #State.Line_inCIP := TRUE; END_IF;
   IF #alwaysON AND NOT #Cmd.Line_CIP_Req THEN #State.Line_inCIP := FALSE; END_IF;
   IF #alwaysON AND #State.Tank_inCIP AND (#IN_LT01 >= #Param.CIP_Ret_ON_SP) THEN
       #State.CIP_ReturnON := TRUE;
   END_IF;
   IF #alwaysON AND (#IN_LT01 <= #Param.CIP_Ret_OFF_SP) THEN #State.CIP_ReturnON := FALSE; END_IF;
END_REGION

REGION Network 12: Loading AV and Pump
   RUNG wire#powerrail
      Contact( #alwaysON )
      wire#w1
      Move(in := #Param.SupplyPump_SP_Speed, out1 => #"OUT_P.03-Speed")
   END_RUNG
   RUNG wire#w1
      Contact( #State.Tank_inloading )
      wire#w2
      S_Coil( #"OUT_AV.10" )
   END_RUNG
   RUNG wire#w2
      Contact( #"IN_FBAV.10" )
      { S7_Templates := "time_type := Time" } #AVinloadTim.TON(pt := T#1s, et =>)
   END_RUNG
   RUNG wire#w2
      Contact( #AVinloadTim.Q )
      S_Coil( #"OUT_P.03" )
   END_RUNG
   RUNG wire#w1
      I_Contact( #State.Tank_inloading )
      wire#w3
      R_Coil( #"OUT_P.03" )
   END_RUNG
   RUNG wire#w3
      { S7_Templates := "time_type := Time" } #SPumpTim.TON(pt := T#5s, et =>)
   END_RUNG
   RUNG wire#w3
      I_Contact( #"IN_FBP.03" )
      Contact( #SPumpTim.Q )
      { S7_Templates := "SrcType := Real" } LE_Contact(in1 := #"IN_P.03-Speed", in2 := 5.0)
      R_Coil( #"OUT_AV.10" )
   END_RUNG
   // the same network as SCL:
   IF #alwaysON THEN #"OUT_P.03-Speed" := #Param.SupplyPump_SP_Speed; END_IF;
   #_w1 := #alwaysON AND #State.Tank_inloading;
   IF #_w1 THEN #"OUT_AV.10" := TRUE; END_IF;
   #AVinloadTim(IN := #_w1 AND #"IN_FBAV.10", PT := T#1s);   // TON
   IF #_w1 AND #AVinloadTim.Q THEN #"OUT_P.03" := TRUE; END_IF;
   #_w2 := #alwaysON AND NOT #State.Tank_inloading;
   IF #_w2 THEN #"OUT_P.03" := FALSE; END_IF;
   #SPumpTim(IN := #_w2, PT := T#5s);   // TON
   IF #_w2 AND NOT #"IN_FBP.03" AND #SPumpTim.Q AND (#"IN_P.03-Speed" <= 5.0) THEN
       #"OUT_AV.10" := FALSE;
   END_IF;
END_REGION

NETWORK
TITLE = Raw Matrial Inload Dose Param
//Sp Dose Qty
      L     #Param.RawDose_SP_Qty;
      T     #Dose.SP_DOSEQTY;
//SP Fine Qty
      L     #Param.RawDose_SP_Qty;
      L     #Param.RawDose_Fine_Qty;
      *R;
      L     100.0;
      /R;
      T     #Dose.SP_FINEQTY;
//SP Stop Qty
      L     #Param.RawDose_Fine_Qty;
      L     #Param.RawDose_Stop_Qty;
      *R;
      L     100.0;
      /R;
      T     #RawDose_Stop_Qty;

//Sp Dose Pump Speed
      L     #Param.RawDose_SP_Speed;
      T     #Dose.SP_COARSESPEED;
//SP Fine Pump Speed
      L     #Param.RawDose_SP_Speed;
      L     #Param.RawDose_Fine_Speed;
      *R;
      L     100.0;
      /R;
      T     #Dose.SP_FINESPEED;
//r_Stop
      L     #Dose.SP_DOSEQTY;
      L     #RawDose_Stop_Qty;
      -R;
      T     #Dose.r_STOP;

REGION Network 14: Raw Matrial Inload Dose Start Cmd
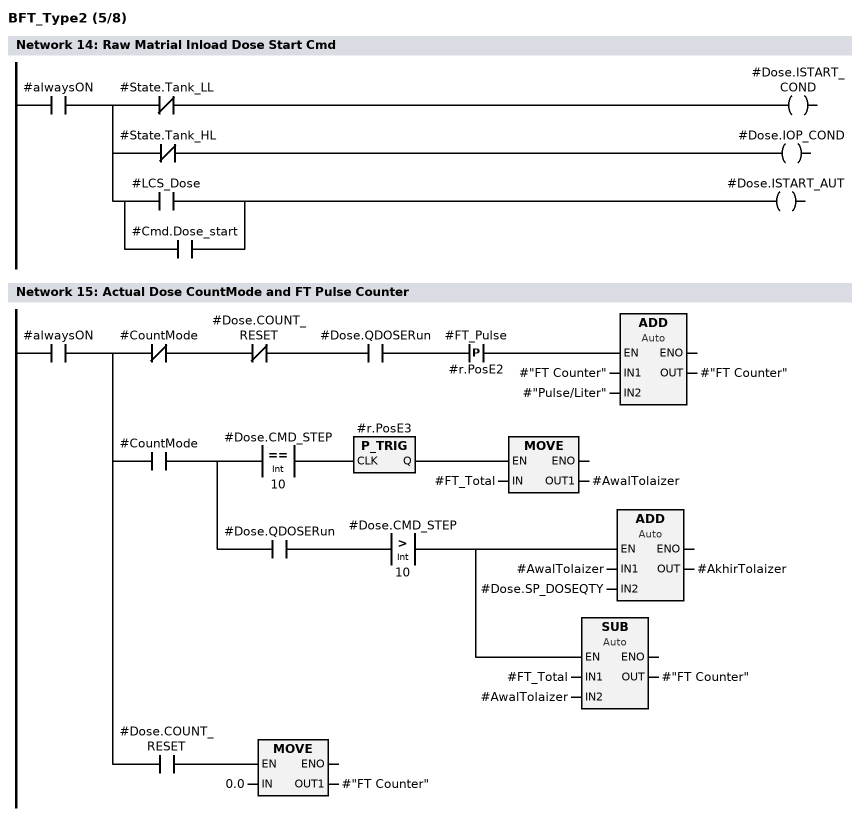
   RUNG wire#powerrail
      Contact( #alwaysON )
      wire#w1
      I_Contact( #State.Tank_LL )
      Coil( #Dose.ISTART_COND )
   END_RUNG
   RUNG wire#w1
      I_Contact( #State.Tank_HL )
      Coil( #Dose.IOP_COND )
   END_RUNG
   RUNG wire#w1
      Contact( #LCS_Dose )
      wire#w2
      Coil( #Dose.ISTART_AUT )
   END_RUNG
   RUNG wire#w1
      Contact( #Cmd.Dose_start )
   END_RUNG wire#w2
   // the same network as SCL:
   #Dose.ISTART_COND := #alwaysON AND NOT #State.Tank_LL;
   #Dose.IOP_COND := #alwaysON AND NOT #State.Tank_HL;
   #Dose.ISTART_AUT := #alwaysON AND (#LCS_Dose OR #Cmd.Dose_start);
END_REGION

REGION Network 15: Actual Dose CountMode and FT Pulse Counter
   RUNG wire#powerrail
      Contact( #alwaysON )
      wire#w1
      I_Contact( #CountMode )
      I_Contact( #Dose.COUNT_RESET )
      Contact( #Dose.QDOSERun )
      P_Contact(operand := #FT_Pulse, bit := #r.PosE2)
      Add(in1 := #"FT Counter", in2 := #"Pulse/Liter", out => #"FT Counter")
   END_RUNG
   RUNG wire#w1
      Contact( #CountMode )
      wire#w2
      { S7_Templates := "SrcType := Int" } EQ_Contact(in1 := #Dose.CMD_STEP, in2 := 10)
      P_Trig( #r.PosE3 )
      Move(in := #FT_Total, out1 => #AwalTolaizer)
   END_RUNG
   RUNG wire#w2
      Contact( #Dose.QDOSERun )
      { S7_Templates := "SrcType := Int" } GT_Contact(in1 := #Dose.CMD_STEP, in2 := 10)
      wire#w3
      Add(in1 := #AwalTolaizer, in2 := #Dose.SP_DOSEQTY, out => #AkhirTolaizer)
   END_RUNG
   RUNG wire#w3
      Sub(in1 := #FT_Total, in2 := #AwalTolaizer, out => #"FT Counter")
   END_RUNG
   RUNG wire#w1
      Contact( #Dose.COUNT_RESET )
      Move(in := 0.0, out1 => #"FT Counter")
   END_RUNG
   // the same network as SCL:
   #_w1 := #alwaysON AND NOT #CountMode AND NOT #Dose.COUNT_RESET AND #Dose.QDOSERun AND #FT_Pulse AND NOT #r.PosE2;   // rising edge of #FT_Pulse
   #r.PosE2 := #FT_Pulse;
   IF #_w1 THEN #"FT Counter" := #"FT Counter" + #"Pulse/Liter"; END_IF;
   #_w2 := #alwaysON AND #CountMode;
   #_w3 := #_w2 AND (#Dose.CMD_STEP = 10);
   #_w4 := #_w3 AND NOT #r.PosE3;   // rising edge
   #r.PosE3 := #_w3;
   IF #_w4 THEN #AwalTolaizer := #FT_Total; END_IF;
   IF #_w2 AND #Dose.QDOSERun AND (#Dose.CMD_STEP > 10) THEN
       #AkhirTolaizer := #AwalTolaizer + #Dose.SP_DOSEQTY;
       #"FT Counter" := #FT_Total - #AwalTolaizer;
   END_IF;
   IF #alwaysON AND #Dose.COUNT_RESET THEN #"FT Counter" := 0.0; END_IF;
END_REGION

REGION Network 16: Raw Matrial Inload Dose
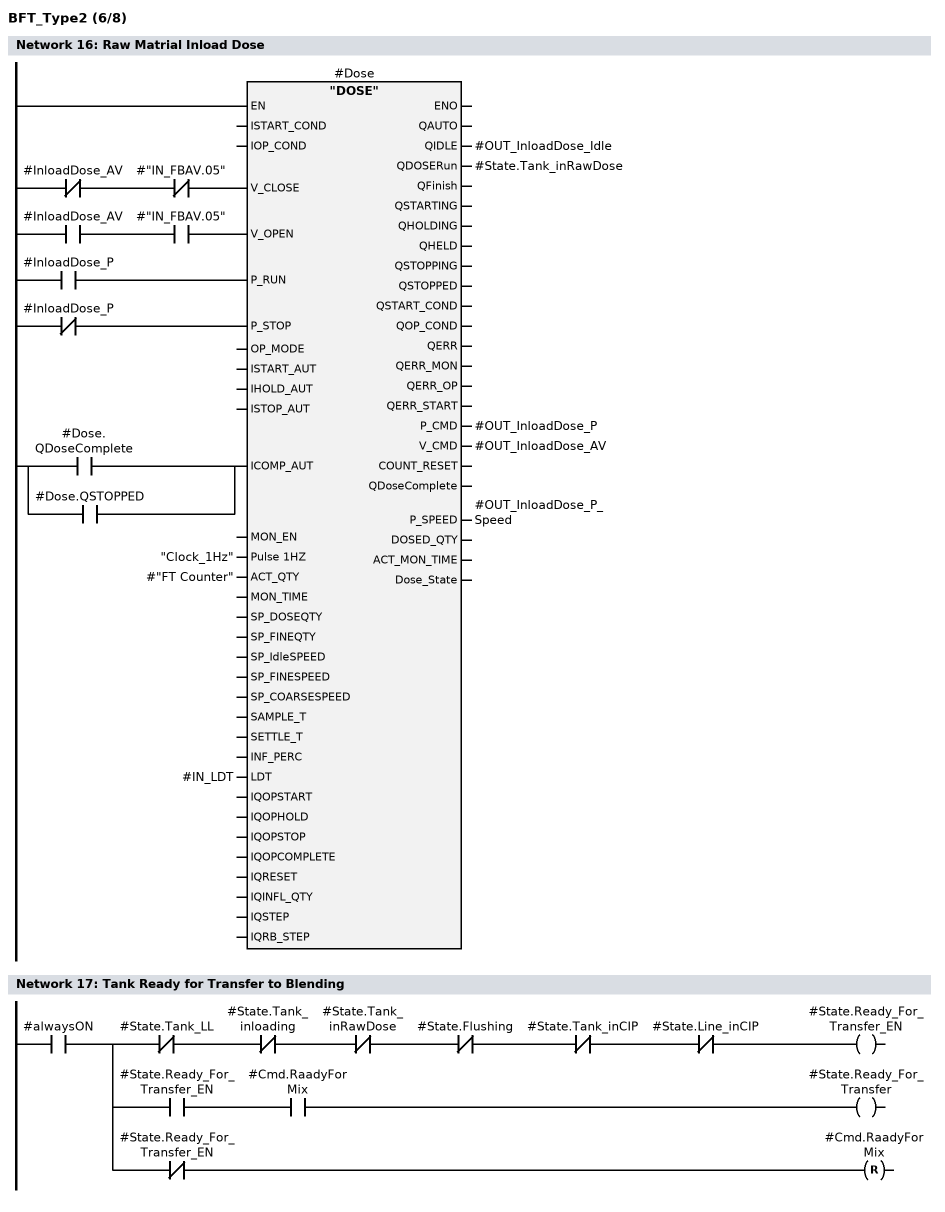
   RUNG wire#powerrail
      #Dose(V_CLOSE := wire#w1, V_OPEN := wire#w2, P_RUN := wire#w3, P_STOP := wire#w4, ICOMP_AUT := wire#w5, ISTART_COND :=, IOP_COND :=, OP_MODE :=, ISTART_AUT :=, IHOLD_AUT :=, ISTOP_AUT :=, MON_EN :=, "Pulse 1HZ" := "Clock_1Hz", ACT_QTY := #"FT Counter", MON_TIME :=, SP_DOSEQTY :=, SP_FINEQTY :=, SP_FINESPEED :=, SP_COARSESPEED :=, SAMPLE_T :=, SETTLE_T :=, INF_PERC :=, LDT := #IN_LDT, IQOPSTART :=, IQOPHOLD :=, IQOPSTOP :=, IQOPCOMPLETE :=, IQRESET :=, IQINFL_QTY :=, IQSTEP :=, IQRB_STEP :=, QAUTO =>, QIDLE => #OUT_InloadDose_Idle, QDOSERun => #State.Tank_inRawDose, QFinish =>, QSTARTING =>, QHOLDING =>, QHELD =>, QSTOPPING =>, QSTOPPED =>, QSTART_COND =>, QOP_COND =>, QERR =>, QERR_MON =>, QERR_OP =>, QERR_START =>, P_CMD => #OUT_InloadDose_P, V_CMD => #OUT_InloadDose_AV, COUNT_RESET =>, QDoseComplete =>, P_SPEED => #OUT_InloadDose_P_Speed, DOSED_QTY =>, ACT_MON_TIME =>, SP_IdleSPEED :=, Dose_State =>)
   END_RUNG
   RUNG wire#powerrail
      I_Contact( #InloadDose_AV )
      I_Contact( #"IN_FBAV.05" )
   END_RUNG wire#w1
   RUNG wire#powerrail
      Contact( #InloadDose_AV )
      Contact( #"IN_FBAV.05" )
   END_RUNG wire#w2
   RUNG wire#powerrail
      Contact( #InloadDose_P )
   END_RUNG wire#w3
   RUNG wire#powerrail
      I_Contact( #InloadDose_P )
   END_RUNG wire#w4
   RUNG wire#powerrail
      Contact( #Dose.QDoseComplete )
   END_RUNG wire#w5
   RUNG wire#powerrail
      Contact( #Dose.QSTOPPED )
   END_RUNG wire#w5
   // the same network as SCL:
   #Dose(V_CLOSE := NOT #InloadDose_AV AND NOT #"IN_FBAV.05",   // "DOSE"
         V_OPEN := #InloadDose_AV AND #"IN_FBAV.05",
         P_RUN := #InloadDose_P,
         P_STOP := NOT #InloadDose_P,
         ICOMP_AUT := #Dose.QDoseComplete OR #Dose.QSTOPPED,
         "Pulse 1HZ" := "Clock_1Hz",
         ACT_QTY := #"FT Counter",
         LDT := #IN_LDT,
         QIDLE => #OUT_InloadDose_Idle,
         QDOSERun => #State.Tank_inRawDose,
         P_CMD => #OUT_InloadDose_P,
         V_CMD => #OUT_InloadDose_AV,
         P_SPEED => #OUT_InloadDose_P_Speed);
END_REGION

REGION Network 17: Tank Ready for Transfer to Blending
   RUNG wire#powerrail
      Contact( #alwaysON )
      wire#w1
      I_Contact( #State.Tank_LL )
      I_Contact( #State.Tank_inloading )
      I_Contact( #State.Tank_inRawDose )
      I_Contact( #State.Flushing )
      I_Contact( #State.Tank_inCIP )
      I_Contact( #State.Line_inCIP )
      Coil( #State.Ready_For_Transfer_EN )
   END_RUNG
   RUNG wire#w1
      Contact( #State.Ready_For_Transfer_EN )
      Contact( #Cmd.RaadyForMix )
      Coil( #State.Ready_For_Transfer )
   END_RUNG
   RUNG wire#w1
      I_Contact( #State.Ready_For_Transfer_EN )
      R_Coil( #Cmd.RaadyForMix )
   END_RUNG
   // the same network as SCL:
   #State.Ready_For_Transfer_EN := #alwaysON AND NOT #State.Tank_LL AND NOT #State.Tank_inloading AND NOT #State.Tank_inRawDose AND NOT #State.Flushing AND NOT #State.Tank_inCIP AND NOT #State.Line_inCIP;
   #State.Ready_For_Transfer := #alwaysON AND #State.Ready_For_Transfer_EN AND #Cmd.RaadyForMix;
   IF #alwaysON AND NOT #State.Ready_For_Transfer_EN THEN #Cmd.RaadyForMix := FALSE; END_IF;
END_REGION

REGION Network 18: Agitator
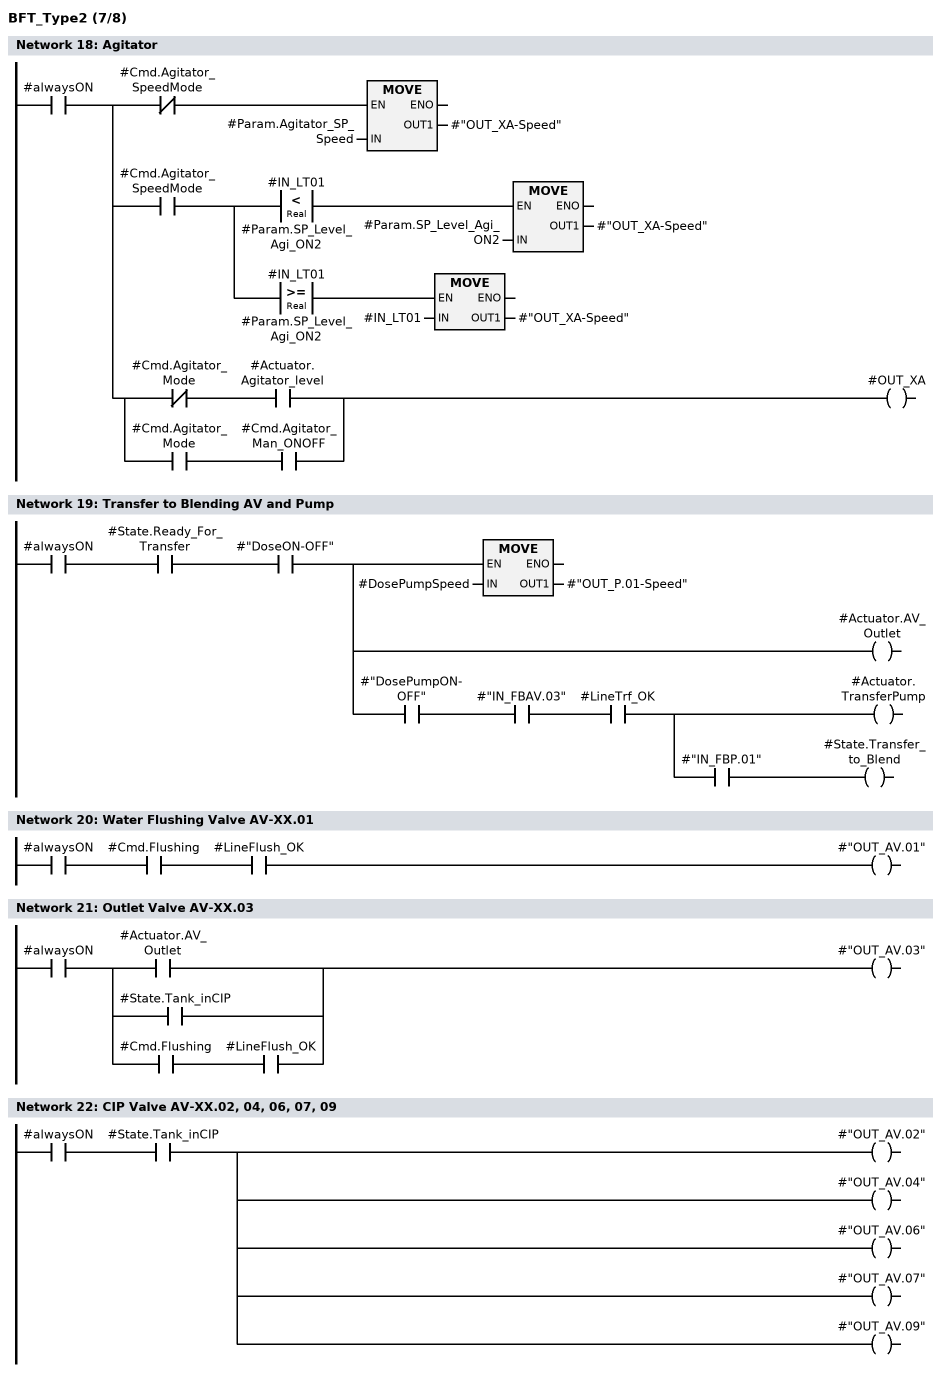
   RUNG wire#powerrail
      Contact( #alwaysON )
      wire#w1
      I_Contact( #Cmd.Agitator_SpeedMode )
      Move(in := #Param.Agitator_SP_Speed, out1 => #"OUT_XA-Speed")
   END_RUNG
   RUNG wire#w1
      Contact( #Cmd.Agitator_SpeedMode )
      wire#w2
      { S7_Templates := "SrcType := Real" } LT_Contact(in1 := #IN_LT01, in2 := #Param.SP_Level_Agi_ON2)
      Move(in := #Param.SP_Level_Agi_ON2, out1 => #"OUT_XA-Speed")
   END_RUNG
   RUNG wire#w2
      { S7_Templates := "SrcType := Real" } GE_Contact(in1 := #IN_LT01, in2 := #Param.SP_Level_Agi_ON2)
      Move(in := #IN_LT01, out1 => #"OUT_XA-Speed")
   END_RUNG
   RUNG wire#w1
      I_Contact( #Cmd.Agitator_Mode )
      Contact( #Actuator.Agitator_level )
      wire#w3
      Coil( #OUT_XA )
   END_RUNG
   RUNG wire#w1
      Contact( #Cmd.Agitator_Mode )
      Contact( #Cmd.Agitator_Man_ONOFF )
   END_RUNG wire#w3
   // the same network as SCL:
   IF #alwaysON AND NOT #Cmd.Agitator_SpeedMode THEN #"OUT_XA-Speed" := #Param.Agitator_SP_Speed; END_IF;
   #_w1 := #alwaysON AND #Cmd.Agitator_SpeedMode;
   IF #_w1 AND (#IN_LT01 < #Param.SP_Level_Agi_ON2) THEN #"OUT_XA-Speed" := #Param.SP_Level_Agi_ON2; END_IF;
   IF #_w1 AND (#IN_LT01 >= #Param.SP_Level_Agi_ON2) THEN #"OUT_XA-Speed" := #IN_LT01; END_IF;
   #OUT_XA := #alwaysON AND ((NOT #Cmd.Agitator_Mode AND #Actuator.Agitator_level) OR (#Cmd.Agitator_Mode AND #Cmd.Agitator_Man_ONOFF));
END_REGION

REGION Network 19: Transfer to Blending AV and Pump
   RUNG wire#powerrail
      Contact( #alwaysON )
      Contact( #State.Ready_For_Transfer )
      Contact( #"DoseON-OFF" )
      wire#w1
      Move(in := #DosePumpSpeed, out1 => #"OUT_P.01-Speed")
   END_RUNG
   RUNG wire#w1
      Coil( #Actuator.AV_Outlet )
   END_RUNG
   RUNG wire#w1
      Contact( #"DosePumpON-OFF" )
      Contact( #"IN_FBAV.03" )
      Contact( #LineTrf_OK )
      wire#w2
      Coil( #Actuator.TransferPump )
   END_RUNG
   RUNG wire#w2
      Contact( #"IN_FBP.01" )
      Coil( #State.Transfer_to_Blend )
   END_RUNG
   // the same network as SCL:
   #_w1 := #alwaysON AND #State.Ready_For_Transfer AND #"DoseON-OFF";
   IF #_w1 THEN #"OUT_P.01-Speed" := #DosePumpSpeed; END_IF;
   #Actuator.AV_Outlet := #_w1;
   #Actuator.TransferPump := #_w1 AND #"DosePumpON-OFF" AND #"IN_FBAV.03" AND #LineTrf_OK;
   #State.Transfer_to_Blend := #Actuator.TransferPump AND #"IN_FBP.01";
END_REGION

REGION Network 20: Water Flushing Valve AV-XX.01
   RUNG wire#powerrail
      Contact( #alwaysON )
      Contact( #Cmd.Flushing )
      Contact( #LineFlush_OK )
      Coil( #"OUT_AV.01" )
   END_RUNG
   // the same network as SCL:
   #"OUT_AV.01" := #alwaysON AND #Cmd.Flushing AND #LineFlush_OK;
END_REGION

REGION Network 21: Outlet Valve AV-XX.03
   RUNG wire#powerrail
      Contact( #alwaysON )
      wire#w1
      Contact( #Actuator.AV_Outlet )
      wire#w2
      Coil( #"OUT_AV.03" )
   END_RUNG
   RUNG wire#w1
      Contact( #State.Tank_inCIP )
   END_RUNG wire#w2
   RUNG wire#w1
      Contact( #Cmd.Flushing )
      Contact( #LineFlush_OK )
   END_RUNG wire#w2
   // the same network as SCL:
   #"OUT_AV.03" := #alwaysON AND (#Actuator.AV_Outlet OR #State.Tank_inCIP OR (#Cmd.Flushing AND #LineFlush_OK));
END_REGION

REGION Network 22: CIP Valve AV-XX.02, 04, 06, 07, 09
   RUNG wire#powerrail
      Contact( #alwaysON )
      Contact( #State.Tank_inCIP )
      wire#w1
      Coil( #"OUT_AV.02" )
   END_RUNG
   RUNG wire#w1
      Coil( #"OUT_AV.04" )
   END_RUNG
   RUNG wire#w1
      Coil( #"OUT_AV.06" )
   END_RUNG
   RUNG wire#w1
      Coil( #"OUT_AV.07" )
   END_RUNG
   RUNG wire#w1
      Coil( #"OUT_AV.09" )
   END_RUNG
   // the same network as SCL:
   #"OUT_AV.02" := #alwaysON AND #State.Tank_inCIP;
   #"OUT_AV.04" := #"OUT_AV.02";
   #"OUT_AV.06" := #"OUT_AV.02";
   #"OUT_AV.07" := #"OUT_AV.02";
   #"OUT_AV.09" := #"OUT_AV.02";
END_REGION

REGION Network 23: Raw Material Inlet Valve AV-XX.05
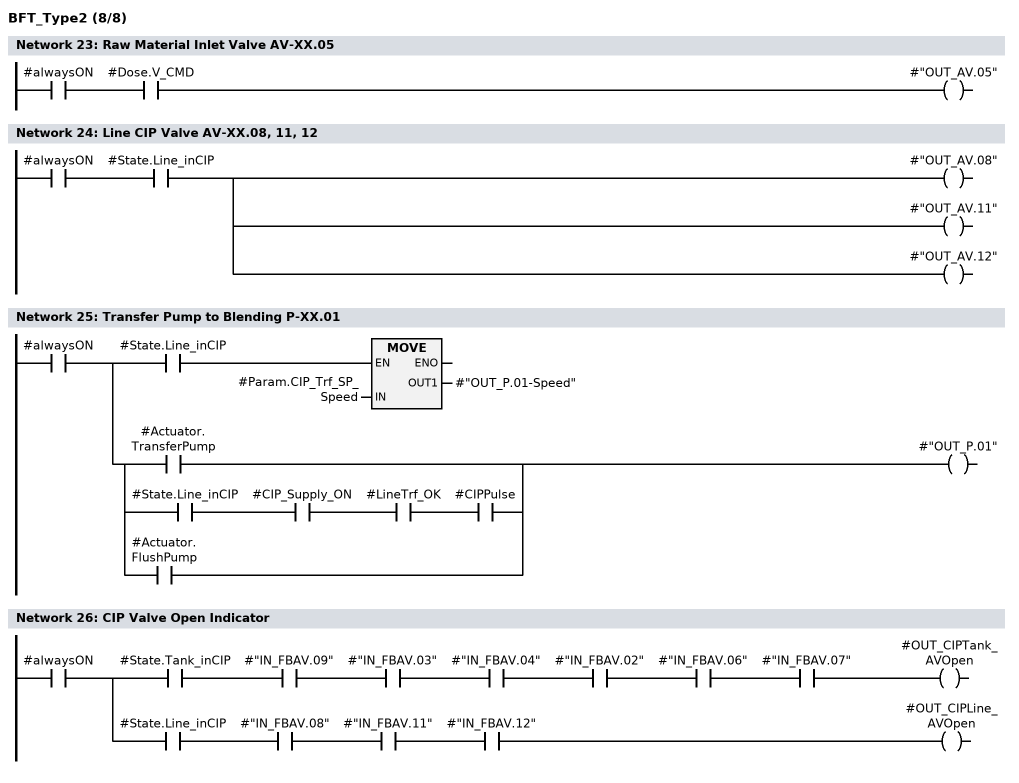
   RUNG wire#powerrail
      Contact( #alwaysON )
      Contact( #Dose.V_CMD )
      Coil( #"OUT_AV.05" )
   END_RUNG
   // the same network as SCL:
   #"OUT_AV.05" := #alwaysON AND #Dose.V_CMD;
END_REGION

REGION Network 24: Line CIP Valve AV-XX.08, 11, 12
   RUNG wire#powerrail
      Contact( #alwaysON )
      Contact( #State.Line_inCIP )
      wire#w1
      Coil( #"OUT_AV.08" )
   END_RUNG
   RUNG wire#w1
      Coil( #"OUT_AV.11" )
   END_RUNG
   RUNG wire#w1
      Coil( #"OUT_AV.12" )
   END_RUNG
   // the same network as SCL:
   #"OUT_AV.08" := #alwaysON AND #State.Line_inCIP;
   #"OUT_AV.11" := #"OUT_AV.08";
   #"OUT_AV.12" := #"OUT_AV.08";
END_REGION

REGION Network 25: Transfer Pump to Blending P-XX.01
   RUNG wire#powerrail
      Contact( #alwaysON )
      wire#w1
      Contact( #State.Line_inCIP )
      Move(in := #Param.CIP_Trf_SP_Speed, out1 => #"OUT_P.01-Speed")
   END_RUNG
   RUNG wire#w1
      Contact( #Actuator.TransferPump )
      wire#w2
      Coil( #"OUT_P.01" )
   END_RUNG
   RUNG wire#w1
      Contact( #State.Line_inCIP )
      Contact( #CIP_Supply_ON )
      Contact( #LineTrf_OK )
      Contact( #CIPPulse )
   END_RUNG wire#w2
   RUNG wire#w1
      Contact( #Actuator.FlushPump )
   END_RUNG wire#w2
   // the same network as SCL:
   IF #alwaysON AND #State.Line_inCIP THEN #"OUT_P.01-Speed" := #Param.CIP_Trf_SP_Speed; END_IF;
   #"OUT_P.01" := #alwaysON AND (#Actuator.TransferPump OR (#State.Line_inCIP AND #CIP_Supply_ON AND #LineTrf_OK AND #CIPPulse) OR #Actuator.FlushPump);
END_REGION

REGION Network 26: CIP Valve Open Indicator
   RUNG wire#powerrail
      Contact( #alwaysON )
      wire#w1
      Contact( #State.Tank_inCIP )
      Contact( #"IN_FBAV.09" )
      Contact( #"IN_FBAV.03" )
      Contact( #"IN_FBAV.04" )
      Contact( #"IN_FBAV.02" )
      Contact( #"IN_FBAV.06" )
      Contact( #"IN_FBAV.07" )
      Coil( #OUT_CIPTank_AVOpen )
   END_RUNG
   RUNG wire#w1
      Contact( #State.Line_inCIP )
      Contact( #"IN_FBAV.08" )
      Contact( #"IN_FBAV.11" )
      Contact( #"IN_FBAV.12" )
      Coil( #OUT_CIPLine_AVOpen )
   END_RUNG
   // the same network as SCL:
   #OUT_CIPTank_AVOpen := #alwaysON AND #State.Tank_inCIP AND #"IN_FBAV.09" AND #"IN_FBAV.03" AND #"IN_FBAV.04" AND #"IN_FBAV.02" AND #"IN_FBAV.06" AND #"IN_FBAV.07";
   #OUT_CIPLine_AVOpen := #alwaysON AND #State.Line_inCIP AND #"IN_FBAV.08" AND #"IN_FBAV.11" AND #"IN_FBAV.12";
END_REGION
END_FUNCTION_BLOCK
